FUNCTION_BLOCK FB_Subscriber IMPLEMENTS I_Subscriber
VAR_INPUT
END_VAR
VAR_OUTPUT
END_VAR
VAR
	_sName				: STRING;
	_sPublisherContent	: STRING;
END_VAR

//FB_Init is always available implicitly and it is used primarily for initialization.
//The return value is not evaluated. For a specific influence, you can also declare the
//methods explicitly and provide additional code there with the standard initialization
//code. You can evaluate the return value.
METHOD FB_Init: BOOL
VAR_INPUT
    bInitRetains: BOOL; // TRUE: the retain variables are initialized (reset warm / reset cold)
    bInCopyCode: BOOL;  // TRUE: the instance will be copied to the copy code afterward (online change)
	sName	: STRING;   
END_VAR
_sName := sName;
END_METHOD

METHOD update : BOOL
VAR_INPUT
	in_sContent			: STRING;
END_VAR
ADSLOGSTR(msgCtrlMask:= ADSLOG_MSGTYPE_ERROR, msgFmtStr:= 'Hey its me %s, i got noftiyed with fresh new content', strArg:= _sName);
_sPublisherContent := in_sContent;
END_METHOD

END_FUNCTION_BLOCK

(* stored: Version 1.1.0.1
   POU FB_Subscriber: Id {70c40a34-d894-42f5-bdf0-8fb2f84ec1fe}, SpecialFunc None
   Method FB_Init: Id {1d6f0229-85cf-403a-80bf-ab8a41e70fca}
   Method update: Id {494fcd53-ba52-49d9-a260-440222b95e61} *)
